FUNCTION F_SCANNER_LightingIntensity : INT
VAR_INPUT
	nUnitLightingIntensity		:INT;
END_VAR

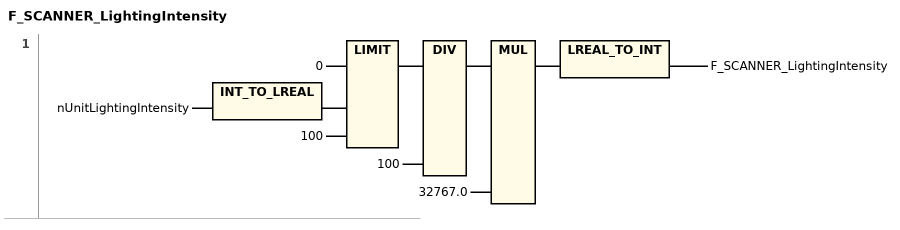
// NETWORK 1
F_SCANNER_LightingIntensity := LREAL_TO_INT((LIMIT(0, INT_TO_LREAL(nUnitLightingIntensity), 100) / 100) * 32767.0);

END_FUNCTION

(* stored: Version 1.1.0.1, ProductVersion 3.1.4024.15
   POU F_SCANNER_LightingIntensity: Id {0963a00e-5c3a-4cf6-ae64-f5d59c9b61ed}, SpecialFunc None *)
